FUNCTION F_DfiNowString : STRING(23)
VAR_INPUT
END_VAR
VAR
	fbGetSystemTime : Tc2_Utilities.GETSYSTEMTIME;
	ft              : T_FILETIME;
	tmst            : TIMESTRUCT;
	nYear : INT;
	nMon  : INT;
	nDay  : INT;
	nHour : INT;
	nMin  : INT;
	nSec  : INT;
	nMs   : INT;
	sYear : STRING(4);
	sMon  : STRING(2);
	sDay  : STRING(2);
	sHour : STRING(2);
	sMin  : STRING(2);
	sSec  : STRING(2);
	sMs   : STRING(3);
END_VAR

// Retorna o instante atual como 'YYYY-MM-DD HH:MM:SS.mmm' (23 chars). Fonte: Tc2_Utilities.GETSYSTEMTIME + FILETIME_TO_SYSTEMTIME (UTC).
// TODO: local timezone conversion (RT Linux timedatectl sets TZ; verify UTC vs local at bench)
fbGetSystemTime(timeLoDW => ft.dwLowDateTime, timeHiDW => ft.dwHighDateTime);
// FILETIME_TO_SYSTEMTIME e FUNCTION: a saida precisa ser capturada (=> tmst),
// senao tmst fica zerado e o timestamp vira '0000-00-00 00:00:00.000'.
// Confirmar no XAE (F2) o nome do parametro de saida: 'systemTime' ou 'pSystemTime'
// (se for POINTER TO TIMESTRUCT, usar: FILETIME_TO_SYSTEMTIME(fileTime := ft, pSystemTime := ADR(tmst));).
FILETIME_TO_SYSTEMTIME(fileTime := ft, systemTime => tmst);

nYear := TO_INT(tmst.wYear);
nMon  := TO_INT(tmst.wMonth);
nDay  := TO_INT(tmst.wDay);
nHour := TO_INT(tmst.wHour);
nMin  := TO_INT(tmst.wMinute);
nSec  := TO_INT(tmst.wSecond);
nMs   := TO_INT(tmst.wMilliseconds);

sYear := INT_TO_STRING(nYear);

IF nMon < 10 THEN sMon := CONCAT('0', INT_TO_STRING(nMon)); ELSE sMon := INT_TO_STRING(nMon); END_IF
IF nDay < 10 THEN sDay := CONCAT('0', INT_TO_STRING(nDay)); ELSE sDay := INT_TO_STRING(nDay); END_IF
IF nHour < 10 THEN sHour := CONCAT('0', INT_TO_STRING(nHour)); ELSE sHour := INT_TO_STRING(nHour); END_IF
IF nMin < 10 THEN sMin := CONCAT('0', INT_TO_STRING(nMin)); ELSE sMin := INT_TO_STRING(nMin); END_IF
IF nSec < 10 THEN sSec := CONCAT('0', INT_TO_STRING(nSec)); ELSE sSec := INT_TO_STRING(nSec); END_IF

IF nMs < 10 THEN
	sMs := CONCAT('00', INT_TO_STRING(nMs));
ELSIF nMs < 100 THEN
	sMs := CONCAT('0', INT_TO_STRING(nMs));
ELSE
	sMs := INT_TO_STRING(nMs);
END_IF

F_DfiNowString := CONCAT(sYear, '-');
F_DfiNowString := CONCAT(F_DfiNowString, sMon);
F_DfiNowString := CONCAT(F_DfiNowString, '-');
F_DfiNowString := CONCAT(F_DfiNowString, sDay);
F_DfiNowString := CONCAT(F_DfiNowString, ' ');
F_DfiNowString := CONCAT(F_DfiNowString, sHour);
F_DfiNowString := CONCAT(F_DfiNowString, ':');
F_DfiNowString := CONCAT(F_DfiNowString, sMin);
F_DfiNowString := CONCAT(F_DfiNowString, ':');
F_DfiNowString := CONCAT(F_DfiNowString, sSec);
F_DfiNowString := CONCAT(F_DfiNowString, '.');
F_DfiNowString := CONCAT(F_DfiNowString, sMs);

END_FUNCTION

(* stored: Version 1.1.0.1
   POU F_DfiNowString: Id {e78f4122-21c3-4f6e-9386-77b892d73e6e}, SpecialFunc None *)
